(* IEC 61131-3 sources: Snap7/Sharp7/LAP_2018_4_Niveauregelung/ConfigTests/Niveauregelung_1, 1 file *)

(* ---- testProgramm.st ---- *)
FUNCTION_BLOCK TestProgramm
VAR_INPUT
END_VAR
VAR_OUTPUT
END_VAR
VAR
    ZyklusAktiv: BOOL;
	Zeit: TON;
END_VAR

(*  *********************************************************** *)
(*  LAP 2018/4 Niveauregelung                                   *)
(*  *********************************************************** *)
